// TIA Portal V17 export
// export: Created 2023-04-11T09:33:27.5010094Z, ExportSetting WithDefaults, DisplayName Totally Integrated Automation Portal, DisplayVersion V17 Update 3, DisplayName TIA Portal Openness, DisplayVersion V17 Update 3, DisplayName TIA Portal Version Control Interface, DisplayVersion V17, DisplayName SINAMICS Startdrive Advanced, DisplayVersion V17 Update2, DisplayName SINAMICS Startdrive G130, G150, S120, S150, SINAMICS MV, S210, DisplayVersion V17 Update2, DisplayName SINAMICS Startdrive G110M, G120, G120C, G120D, G120P, G115D, DisplayVersion V17 Update2, DisplayName STEP 7 Professional, DisplayVersion V17 Update 3, DisplayName STEP 7 Safety, DisplayVersion V17, DisplayName WinCC UA Professional, DisplayVersion V17 Update 3
FUNCTION_BLOCK "FB_coverControl"   // FB20, LAD
TITLE = Standart cylinder control
{ S7_Optimized_Access := 'TRUE' }
VERSION : 0.1
// stored: AutoNumber true, IsIECCheckEnabled false, IsRetainMemResEnabled false, MemoryReserve 100, SetENOAutomatically false, UDAEnableTagReadback false
   VAR_INPUT
      Request_UP : Bool;
      Request_Down : Bool;
      Sensor_Lock : Bool;
      Sensor_UP : Bool;
      With_UP : Bool;
      Sensor_Down : Bool;
      With_Down : Bool;
      Enable_UP : Bool;
      Enable_Down : Bool;
      ErrorMonitoring : Bool;
      UnlockManual : Bool;
      ManualControlActive : Bool;
      SensorDelay_Up : Time;
      TimeForError_A : Time;
      TimeForError_B : Time;
   END_VAR
   VAR_OUTPUT
      Out_UP : Bool;
      Out_Down : Bool;
      Out_Unlock : Bool;
      Done_LockDown : Bool;
      Done_Up : Bool;
      Done_Down : Bool;
      Error_LockDown : Bool;
      Error_Up : Bool;
      Error_Down : Bool;
   END_VAR
   VAR
      FB_FaultModule_Instance { S7_SetPoint := 'True'} : "FB_faultModule";
      IEC_Timer_0_Instance { S7_SetPoint := 'True'} : TON_TIME;
      IEC_Timer_0_Instance_2 { S7_SetPoint := 'True'} : TON_TIME;
      IEC_Timer_0_Instance_3 { S7_SetPoint := 'True'} : TON_TIME;
      IEC_Timer_0_Instance_4 { S7_SetPoint := 'True'} : TON_TIME;
      edge : Array[0..1] of Bool;
      Out_Unlock_temp : Bool;
      IEC_Timer_0_Instance_1 { S7_SetPoint := 'True'} : TON_TIME;
   END_VAR
   VAR_TEMP
      Out_Up_temp : Bool;
      Out_Down_temp : Bool;
   END_VAR
   VAR_TEMP   // added for the SCL form of the ladder/FBD networks
      _w1 : Bool;
   END_VAR
BEGIN

REGION Network 1: OUT UP / UNLOCK
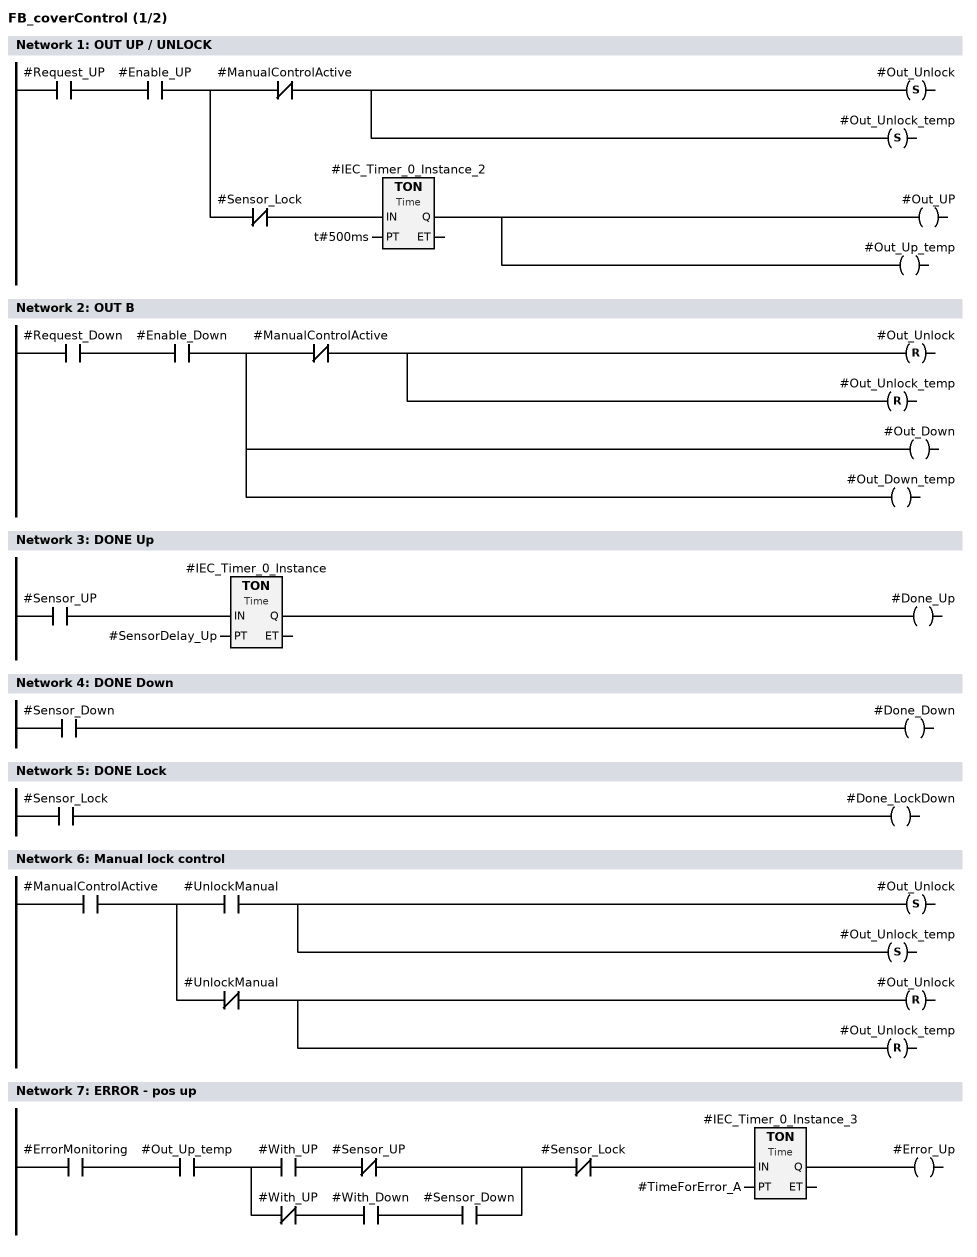
   RUNG wire#powerrail
      Contact( #Request_UP )
      Contact( #Enable_UP )
      wire#w1
      I_Contact( #ManualControlActive )
      wire#w2
      S_Coil( #Out_Unlock )
   END_RUNG
   RUNG wire#w2
      S_Coil( #Out_Unlock_temp )
   END_RUNG
   RUNG wire#w1
      I_Contact( #Sensor_Lock )
      { S7_Templates := "time_type := Time" } #IEC_Timer_0_Instance_2.TON(pt := t#500ms, et =>)
      wire#w3
      Coil( #Out_UP )
   END_RUNG
   RUNG wire#w3
      Coil( #Out_Up_temp )
   END_RUNG
   // the same network as SCL:
   #_w1 := #Request_UP AND #Enable_UP;
   IF #_w1 AND NOT #ManualControlActive THEN
       #Out_Unlock := TRUE;
       #Out_Unlock_temp := TRUE;
   END_IF;
   #IEC_Timer_0_Instance_2(IN := #_w1 AND NOT #Sensor_Lock, PT := t#500ms);   // TON
   #Out_UP := #IEC_Timer_0_Instance_2.Q;
   #Out_Up_temp := #IEC_Timer_0_Instance_2.Q;
END_REGION

REGION Network 2: OUT B
   RUNG wire#powerrail
      Contact( #Request_Down )
      Contact( #Enable_Down )
      wire#w1
      I_Contact( #ManualControlActive )
      wire#w2
      R_Coil( #Out_Unlock )
   END_RUNG
   RUNG wire#w2
      R_Coil( #Out_Unlock_temp )
   END_RUNG
   RUNG wire#w1
      Coil( #Out_Down )
   END_RUNG
   RUNG wire#w1
      Coil( #Out_Down_temp )
   END_RUNG
   // the same network as SCL:
   #_w1 := #Request_Down AND #Enable_Down;
   IF #_w1 AND NOT #ManualControlActive THEN
       #Out_Unlock := FALSE;
       #Out_Unlock_temp := FALSE;
   END_IF;
   #Out_Down := #_w1;
   #Out_Down_temp := #_w1;
END_REGION

REGION Network 3: DONE Up
   RUNG wire#powerrail
      Contact( #Sensor_UP )
      { S7_Templates := "time_type := Time" } #IEC_Timer_0_Instance.TON(pt := #SensorDelay_Up, et =>)
      Coil( #Done_Up )
   END_RUNG
   // the same network as SCL:
   #IEC_Timer_0_Instance(IN := #Sensor_UP, PT := #SensorDelay_Up);   // TON
   #Done_Up := #IEC_Timer_0_Instance.Q;
END_REGION

REGION Network 4: DONE Down
   RUNG wire#powerrail
      Contact( #Sensor_Down )
      Coil( #Done_Down )
   END_RUNG
   // the same network as SCL:
   #Done_Down := #Sensor_Down;
END_REGION

REGION Network 5: DONE Lock
   RUNG wire#powerrail
      Contact( #Sensor_Lock )
      Coil( #Done_LockDown )
   END_RUNG
   // the same network as SCL:
   #Done_LockDown := #Sensor_Lock;
END_REGION

REGION Network 6: Manual lock control
   RUNG wire#powerrail
      Contact( #ManualControlActive )
      wire#w1
      Contact( #UnlockManual )
      wire#w2
      S_Coil( #Out_Unlock )
   END_RUNG
   RUNG wire#w2
      S_Coil( #Out_Unlock_temp )
   END_RUNG
   RUNG wire#w1
      I_Contact( #UnlockManual )
      wire#w3
      R_Coil( #Out_Unlock )
   END_RUNG
   RUNG wire#w3
      R_Coil( #Out_Unlock_temp )
   END_RUNG
   // the same network as SCL:
   IF #ManualControlActive AND #UnlockManual THEN
       #Out_Unlock := TRUE;
       #Out_Unlock_temp := TRUE;
   END_IF;
   IF #ManualControlActive AND NOT #UnlockManual THEN
       #Out_Unlock := FALSE;
       #Out_Unlock_temp := FALSE;
   END_IF;
END_REGION

REGION Network 7: ERROR - pos up
   RUNG wire#powerrail
      Contact( #ErrorMonitoring )
      Contact( #Out_Up_temp )
      wire#w1
      Contact( #With_UP )
      I_Contact( #Sensor_UP )
      wire#w2
      I_Contact( #Sensor_Lock )
      { S7_Templates := "time_type := Time" } #IEC_Timer_0_Instance_3.TON(pt := #TimeForError_A, et =>)
      Coil( #Error_Up )
   END_RUNG
   RUNG wire#w1
      I_Contact( #With_UP )
      Contact( #With_Down )
      Contact( #Sensor_Down )
   END_RUNG wire#w2
   // the same network as SCL:
   #IEC_Timer_0_Instance_3(IN := #ErrorMonitoring AND #Out_Up_temp AND ((#With_UP AND NOT #Sensor_UP) OR (NOT #With_UP AND #With_Down AND #Sensor_Down)) AND NOT #Sensor_Lock,   // TON
                           PT := #TimeForError_A);
   #Error_Up := #IEC_Timer_0_Instance_3.Q;
END_REGION

REGION Network 8: ERROR - pos down
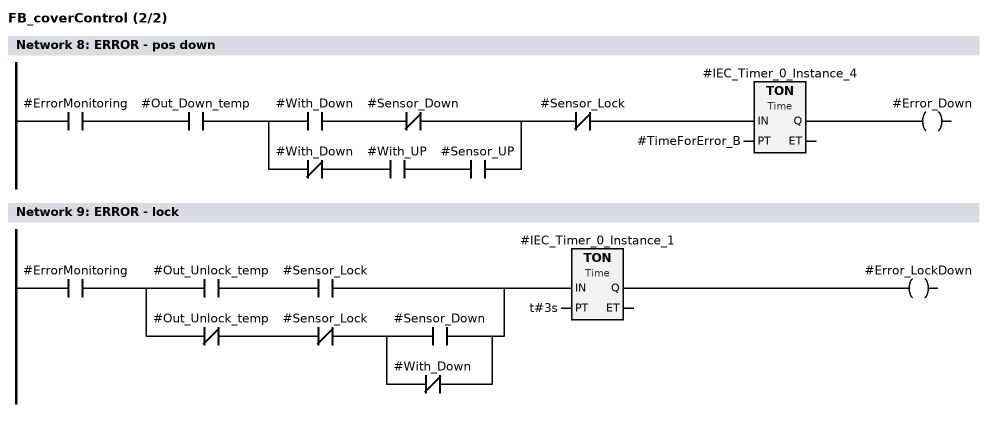
   RUNG wire#powerrail
      Contact( #ErrorMonitoring )
      Contact( #Out_Down_temp )
      wire#w1
      Contact( #With_Down )
      I_Contact( #Sensor_Down )
      wire#w2
      I_Contact( #Sensor_Lock )
      { S7_Templates := "time_type := Time" } #IEC_Timer_0_Instance_4.TON(pt := #TimeForError_B, et =>)
      Coil( #Error_Down )
   END_RUNG
   RUNG wire#w1
      I_Contact( #With_Down )
      Contact( #With_UP )
      Contact( #Sensor_UP )
   END_RUNG wire#w2
   // the same network as SCL:
   #IEC_Timer_0_Instance_4(IN := #ErrorMonitoring AND #Out_Down_temp AND ((#With_Down AND NOT #Sensor_Down) OR (NOT #With_Down AND #With_UP AND #Sensor_UP)) AND NOT #Sensor_Lock,   // TON
                           PT := #TimeForError_B);
   #Error_Down := #IEC_Timer_0_Instance_4.Q;
END_REGION

REGION Network 9: ERROR - lock
   RUNG wire#powerrail
      Contact( #ErrorMonitoring )
      wire#w1
      Contact( #Out_Unlock_temp )
      Contact( #Sensor_Lock )
      wire#w2
      { S7_Templates := "time_type := Time" } #IEC_Timer_0_Instance_1.TON(pt := t#3s, et =>)
      Coil( #Error_LockDown )
   END_RUNG
   RUNG wire#w1
      I_Contact( #Out_Unlock_temp )
      I_Contact( #Sensor_Lock )
      wire#w3
      Contact( #Sensor_Down )
   END_RUNG wire#w2
   RUNG wire#w3
      I_Contact( #With_Down )
   END_RUNG wire#w2
   // the same network as SCL:
   #IEC_Timer_0_Instance_1(IN := #ErrorMonitoring AND ((#Out_Unlock_temp AND #Sensor_Lock) OR (NOT #Out_Unlock_temp AND NOT #Sensor_Lock AND (#Sensor_Down OR NOT #With_Down))),   // TON
                           PT := t#3s);
   #Error_LockDown := #IEC_Timer_0_Instance_1.Q;
END_REGION
END_FUNCTION_BLOCK
